INTERFACE I_GripperModule

END_INTERFACE

(* stored: Version 1.1.0.1, ProductVersion 3.1.4024.12
   Itf I_GripperModule: Id {2bd9185b-99f8-4c7f-ab45-2bb87f682e46} *)
